(* CoDeSys 2.3.9.41 project: RAUMTEMP_REGELUNG.pro *)
(* Libraries: STANDARD.LIB 5.6.98 11:03:02 *)

(* Task configuration *)
TASK Standard (PRIORITY := 0, INTERVAL := T#1ms);
	MAIN
END_TASK

(* Global variable list: Global_Variables *)
VAR_GLOBAL
	(* LEDs *)
	LED_BLUE AT %I* : BOOL;
	LED_GREEN AT %I* : BOOL;
	LED_RED AT %I* : BOOL;
END_VAR
VAR_GLOBAL CONSTANT
	T : REAL := 0.001;
END_VAR

(* Data type *)
TYPE COLOR_T :
(
	BLUE := 1,
	GREEN,
	RED
);
END_TYPE

(* POU MAIN, ST *)
PROGRAM MAIN
VAR
	(* Input *)
	istTempUI AT %I* : UINT;
	(* Local variable *)
	istTempR : REAL;
	(* Output *)
	strHeizventil AT %Q* : UINT;
	(* Regler *)
	reg : TEMP_REGLER;
END_VAR
istTempR := TEMP_SENSOR_CONV(istTempUI);
IF istTempR < 19 THEN
	LED_BLUE := 1;
	LED_GREEN := 0;
	LED_RED := 0;
ELSIF istTempR < 23 THEN
	LED_BLUE := 0;
	LED_GREEN := 1;
	LED_RED := 0;
ELSE
	LED_BLUE := 0;
	LED_GREEN := 0;
	LED_RED := 1;
END_IF
reg(y :=istTempR);
strHeizventil := REAL_TO_UINT(reg.u * 32767 / 100);
END_PROGRAM

(* POU TEMP_REGLER, ST *)
FUNCTION_BLOCK TEMP_REGLER
VAR_INPUT
	y : REAL;
END_VAR
VAR_OUTPUT
	u : REAL;
END_VAR
VAR
	ui : REAL := 0;
END_VAR
ui := ui + T / 3600 * (20 - y);
u := 20 * (20 - y) + ui;
END_FUNCTION_BLOCK

(* POU TEMP_SENSOR_CONV, ST *)
FUNCTION TEMP_SENSOR_CONV : REAL
VAR_INPUT
	temp : UINT;
END_VAR
VAR
END_VAR
TEMP_SENSOR_CONV := UINT_TO_REAL(temp) * 30 / 32767;
END_FUNCTION
